// TIA Portal project "Erronka4" (V15.1)

(* hardware
DEVICE "S7-1200 station_1"  S7-1200 Station
   slot 0: "Rack_0"  S7-1200 Rack  Rack  V1.0
   slot 1: "PLC_1"  CPU 1214C AC/DC/Rly  6ES7 214-1BG40-0XB0  V4.0
   slot 3: "AQ 1x12BIT_1"  AQ1 signal board  6ES7 232-4HA30-0XB0  V1.0
*)

// ===== PLC "PLC_1"  CPU 1214C AC/DC/Rly =====

VAR_GLOBAL   // PLC tag table "Etapas"
   "Etapa0" AT %M16.0 : Bool;
   "Etapa1" AT %M16.1 : Bool;
   "Etapa2" AT %M16.2 : Bool;
   "Etapa3" AT %M16.3 : Bool;
   "Etapa4" AT %M16.4 : Bool;
   "Etapa5" AT %M16.5 : Bool;
   "Etapa6" AT %M16.6 : Bool;
   "Etapa7" AT %M16.7 : Bool;
   "Etapa8" AT %M17.0 : Bool;
   "Etapa9" AT %M17.1 : Bool;
   "Etapa20" AT %M20.0 : Bool;   // Inicio de STOP
   "Etapa21" AT %M20.1 : Bool;   // STOP
   "Etapa22" AT %M20.2 : Bool;   // STOP
   "MRMarca" AT %M90.0 : Bool;
   "Tag_2" AT %M302.0 : Bool;
   "Tag_3" AT %M300.0 : Bool;
   "Tag_4" AT %M300.1 : Bool;
   "Tag_6" AT %M301.0 : Bool;
   "Tag_7" AT %MB302 : Byte;
   "Tag_8" AT %MD16 : DWord;
   "Tag_9" AT %MD90 : DWord;
   "Tag_10" AT %M50.0 : Bool;
   "Tag_12" AT %M50.1 : Bool;
   "Tag_13" AT %MD70 : DWord;   // Tensión para mover MR
   "Tag_14" AT %MD74 : DWord;
   "CONTADORSALIDA" AT %MW100 : Int;
   "MARCAMOTORT" AT %M250.0 : Bool;
   "Tag_1" AT %MD250 : DWord;
END_VAR

VAR_GLOBAL   // PLC tag table "Entradas"
   "SDP1" AT %I0.1 : Bool;
   "SDP2" AT %I0.2 : Bool;
   "SDP3" AT %I0.3 : Bool;
   "SDP4" AT %I0.4 : Bool;
   "M" AT %I0.5 : Bool;
   "PE" AT %I0.6 : Bool;
   "CR0" AT %I0.7 : Bool;
   "CR1" AT %I1.0 : Bool;
   "CT0" AT %I1.1 : Bool;
   "CT1" AT %I1.2 : Bool;
   "CC0" AT %I1.3 : Bool;
   "CC1" AT %I1.4 : Bool;
   "STOP" AT %I0.0 : Bool;
END_VAR

VAR_GLOBAL   // PLC tag table "Salidas"
   "MR" AT %Q2.4 : Bool;
   "ACC" AT %Q0.1 : Bool;
   "DEC" AT %Q0.2 : Bool;
   "CR+" AT %Q0.3 : Bool;
   "CR-" AT %Q0.4 : Bool;
   "CT+" AT %Q0.5 : Bool;
   "CT-" AT %Q0.6 : Bool;
   "CC+" AT %Q0.7 : Bool;
   "CC-" AT %Q1.0 : Bool;
   "MT" AT %Q1.1 : Bool;
   "SEÑAL VARIADOR" AT %Q0.0 : Bool;
   "Tag_16" AT %QW80 : Int;
END_VAR

// folder: System blocks/Program resources

DATA_BLOCK "Temporizador1"   // DB1
{ S7_Optimized_Access := 'TRUE' }
AUTHOR : Simatic
FAMILY : IEC
NAME : IEC_TMR
VERSION : 1.0
// stored: InstanceOfName IEC_TIMER
"IEC_TIMER"
BEGIN
END_DATA_BLOCK

DATA_BLOCK "Contador"   // DB3
{ S7_Optimized_Access := 'TRUE' }
AUTHOR : Simatic
FAMILY : IEC
NAME : CNTR
VERSION : 1.0
// stored: InstanceOfName IEC_COUNTER
"IEC_COUNTER"
BEGIN
END_DATA_BLOCK

// folder: (top level)

FUNCTION "GrafcetPrincipal" : Void   // FC1, LAD
{ S7_Optimized_Access := 'TRUE' }
VERSION : 0.1
   VAR_TEMP   // added for the SCL form of the ladder/FBD networks
      _w1 : Bool;
   END_VAR
BEGIN

REGION Network 1
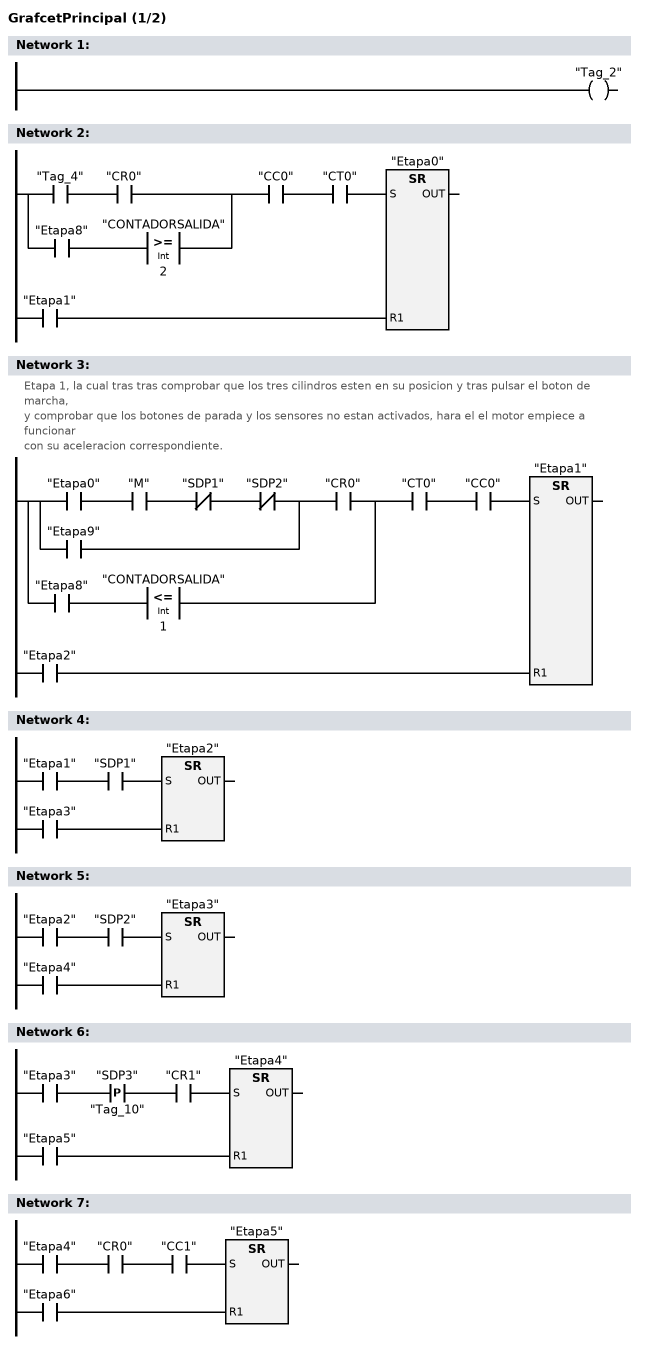
   RUNG wire#powerrail
      Coil( "Tag_2" )
   END_RUNG
   // the same network as SCL:
   "Tag_2" := TRUE;
END_REGION

REGION Network 2
   RUNG wire#powerrail
      Contact( "Tag_4" )
      Contact( "CR0" )
      wire#w1
      Contact( "CC0" )
      Contact( "CT0" )
      S_SR(operand := "Etapa0", r1 := wire#w2)
   END_RUNG
   RUNG wire#powerrail
      Contact( "Etapa8" )
      { S7_Templates := "SrcType := Int" } GE_Contact(in1 := "CONTADORSALIDA", in2 := 2)
   END_RUNG wire#w1
   RUNG wire#powerrail
      Contact( "Etapa1" )
   END_RUNG wire#w2
   // the same network as SCL:
   IF (("Tag_4" AND "CR0") OR ("Etapa8" AND ("CONTADORSALIDA" >= 2))) AND "CC0" AND "CT0" THEN
       "Etapa0" := TRUE;   // SR flip-flop
   END_IF;
   IF "Etapa1" THEN "Etapa0" := FALSE; END_IF;
END_REGION

REGION Network 3
   // Etapa 1, la cual tras tras comprobar que los tres cilindros esten en su posicion y tras pulsar el boton de marcha, 
   // y comprobar que los botones de parada y los sensores no estan activados, hara el el motor empiece a funcionar
   // con su aceleracion correspondiente.
   RUNG wire#powerrail
      Contact( "Etapa0" )
      Contact( "M" )
      I_Contact( "SDP1" )
      I_Contact( "SDP2" )
      wire#w1
      Contact( "CR0" )
      wire#w2
      Contact( "CT0" )
      Contact( "CC0" )
      S_SR(operand := "Etapa1", r1 := wire#w3)
   END_RUNG
   RUNG wire#powerrail
      Contact( "Etapa9" )
   END_RUNG wire#w1
   RUNG wire#powerrail
      Contact( "Etapa8" )
      { S7_Templates := "SrcType := Int" } LE_Contact(in1 := "CONTADORSALIDA", in2 := 1)
   END_RUNG wire#w2
   RUNG wire#powerrail
      Contact( "Etapa2" )
   END_RUNG wire#w3
   // the same network as SCL:
   IF (((("Etapa0" AND "M" AND NOT "SDP1" AND NOT "SDP2") OR "Etapa9") AND "CR0") OR ("Etapa8" AND ("CONTADORSALIDA" <= 1))) AND "CT0" AND "CC0" THEN
       "Etapa1" := TRUE;   // SR flip-flop
   END_IF;
   IF "Etapa2" THEN "Etapa1" := FALSE; END_IF;
END_REGION

REGION Network 4
   RUNG wire#powerrail
      Contact( "Etapa1" )
      Contact( "SDP1" )
      S_SR(operand := "Etapa2", r1 := wire#w1)
   END_RUNG
   RUNG wire#powerrail
      Contact( "Etapa3" )
   END_RUNG wire#w1
   // the same network as SCL:
   IF "Etapa1" AND "SDP1" THEN
       "Etapa2" := TRUE;   // SR flip-flop
   END_IF;
   IF "Etapa3" THEN "Etapa2" := FALSE; END_IF;
END_REGION

REGION Network 5
   RUNG wire#powerrail
      Contact( "Etapa2" )
      Contact( "SDP2" )
      S_SR(operand := "Etapa3", r1 := wire#w1)
   END_RUNG
   RUNG wire#powerrail
      Contact( "Etapa4" )
   END_RUNG wire#w1
   // the same network as SCL:
   IF "Etapa2" AND "SDP2" THEN
       "Etapa3" := TRUE;   // SR flip-flop
   END_IF;
   IF "Etapa4" THEN "Etapa3" := FALSE; END_IF;
END_REGION

REGION Network 6
   RUNG wire#powerrail
      Contact( "Etapa3" )
      P_Contact(operand := "SDP3", bit := "Tag_10")
      Contact( "CR1" )
      S_SR(operand := "Etapa4", r1 := wire#w1)
   END_RUNG
   RUNG wire#powerrail
      Contact( "Etapa5" )
   END_RUNG wire#w1
   // the same network as SCL:
   #_w1 := "Etapa3" AND "SDP3" AND NOT "Tag_10";   // rising edge of "SDP3"
   "Tag_10" := "SDP3";
   IF #_w1 AND "CR1" THEN
       "Etapa4" := TRUE;   // SR flip-flop
   END_IF;
   IF "Etapa5" THEN "Etapa4" := FALSE; END_IF;
END_REGION

REGION Network 7
   RUNG wire#powerrail
      Contact( "Etapa4" )
      Contact( "CR0" )
      Contact( "CC1" )
      S_SR(operand := "Etapa5", r1 := wire#w1)
   END_RUNG
   RUNG wire#powerrail
      Contact( "Etapa6" )
   END_RUNG wire#w1
   // the same network as SCL:
   IF "Etapa4" AND "CR0" AND "CC1" THEN
       "Etapa5" := TRUE;   // SR flip-flop
   END_IF;
   IF "Etapa6" THEN "Etapa5" := FALSE; END_IF;
END_REGION

REGION Network 8
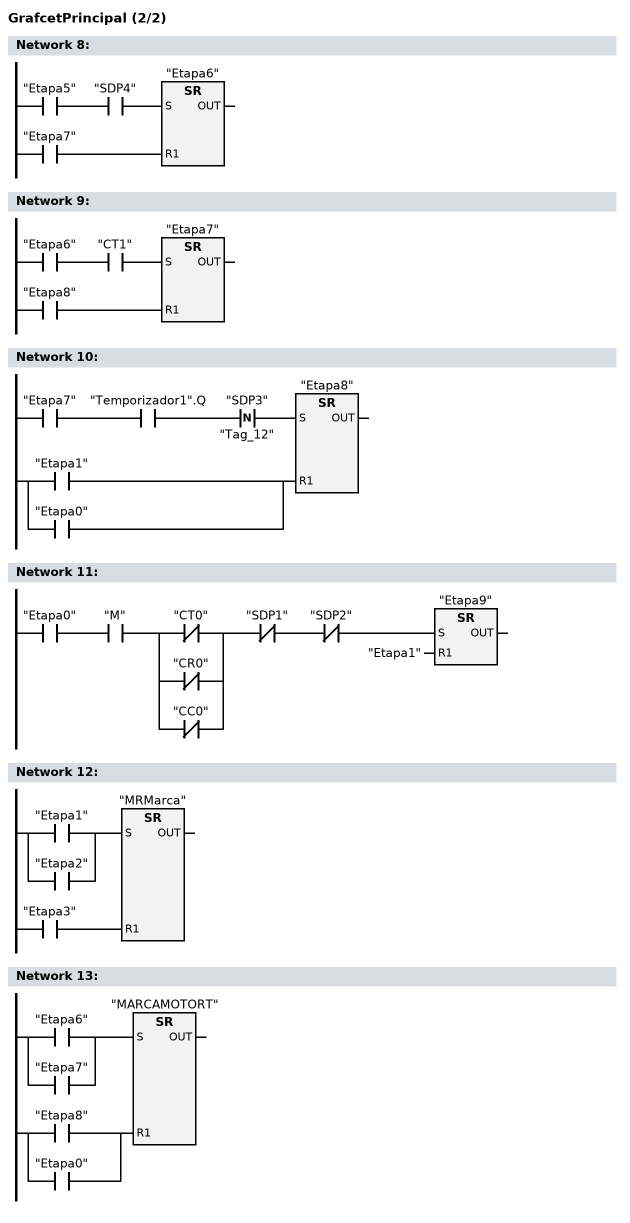
   RUNG wire#powerrail
      Contact( "Etapa5" )
      Contact( "SDP4" )
      S_SR(operand := "Etapa6", r1 := wire#w1)
   END_RUNG
   RUNG wire#powerrail
      Contact( "Etapa7" )
   END_RUNG wire#w1
   // the same network as SCL:
   IF "Etapa5" AND "SDP4" THEN
       "Etapa6" := TRUE;   // SR flip-flop
   END_IF;
   IF "Etapa7" THEN "Etapa6" := FALSE; END_IF;
END_REGION

REGION Network 9
   RUNG wire#powerrail
      Contact( "Etapa6" )
      Contact( "CT1" )
      S_SR(operand := "Etapa7", r1 := wire#w1)
   END_RUNG
   RUNG wire#powerrail
      Contact( "Etapa8" )
   END_RUNG wire#w1
   // the same network as SCL:
   IF "Etapa6" AND "CT1" THEN
       "Etapa7" := TRUE;   // SR flip-flop
   END_IF;
   IF "Etapa8" THEN "Etapa7" := FALSE; END_IF;
END_REGION

REGION Network 10
   RUNG wire#powerrail
      Contact( "Etapa7" )
      Contact( "Temporizador1".Q )
      N_Contact(operand := "SDP3", bit := "Tag_12")
      S_SR(operand := "Etapa8", r1 := wire#w1)
   END_RUNG
   RUNG wire#powerrail
      Contact( "Etapa1" )
   END_RUNG wire#w1
   RUNG wire#powerrail
      Contact( "Etapa0" )
   END_RUNG wire#w1
   // the same network as SCL:
   #_w1 := "Etapa7" AND "Temporizador1".Q AND NOT "SDP3" AND "Tag_12";   // falling edge of "SDP3"
   "Tag_12" := "SDP3";
   IF #_w1 THEN
       "Etapa8" := TRUE;   // SR flip-flop
   END_IF;
   IF "Etapa1" OR "Etapa0" THEN "Etapa8" := FALSE; END_IF;
END_REGION

REGION Network 11
   RUNG wire#powerrail
      Contact( "Etapa0" )
      Contact( "M" )
      wire#w1
      I_Contact( "CT0" )
      wire#w2
      I_Contact( "SDP1" )
      I_Contact( "SDP2" )
      S_SR(operand := "Etapa9", r1 := "Etapa1")
   END_RUNG
   RUNG wire#w1
      I_Contact( "CR0" )
   END_RUNG wire#w2
   RUNG wire#w1
      I_Contact( "CC0" )
   END_RUNG wire#w2
   // the same network as SCL:
   IF "Etapa0" AND "M" AND (NOT "CT0" OR NOT "CR0" OR NOT "CC0") AND NOT "SDP1" AND NOT "SDP2" THEN
       "Etapa9" := TRUE;   // SR flip-flop
   END_IF;
   IF "Etapa1" THEN "Etapa9" := FALSE; END_IF;
END_REGION

REGION Network 12
   RUNG wire#powerrail
      Contact( "Etapa1" )
      wire#w1
      S_SR(operand := "MRMarca", r1 := wire#w2)
   END_RUNG
   RUNG wire#powerrail
      Contact( "Etapa2" )
   END_RUNG wire#w1
   RUNG wire#powerrail
      Contact( "Etapa3" )
   END_RUNG wire#w2
   // the same network as SCL:
   IF "Etapa1" OR "Etapa2" THEN
       "MRMarca" := TRUE;   // SR flip-flop
   END_IF;
   IF "Etapa3" THEN "MRMarca" := FALSE; END_IF;
END_REGION

REGION Network 13
   RUNG wire#powerrail
      Contact( "Etapa6" )
      wire#w1
      S_SR(operand := "MARCAMOTORT", r1 := wire#w2)
   END_RUNG
   RUNG wire#powerrail
      Contact( "Etapa7" )
   END_RUNG wire#w1
   RUNG wire#powerrail
      Contact( "Etapa8" )
   END_RUNG wire#w2
   RUNG wire#powerrail
      Contact( "Etapa0" )
   END_RUNG wire#w2
   // the same network as SCL:
   IF "Etapa6" OR "Etapa7" THEN
       "MARCAMOTORT" := TRUE;   // SR flip-flop
   END_IF;
   IF "Etapa8" OR "Etapa0" THEN "MARCAMOTORT" := FALSE; END_IF;
END_REGION
END_FUNCTION

FUNCTION "ParadaStop" : Void   // FC2, LAD
{ S7_Optimized_Access := 'TRUE' }
VERSION : 0.1
BEGIN

REGION Network 1
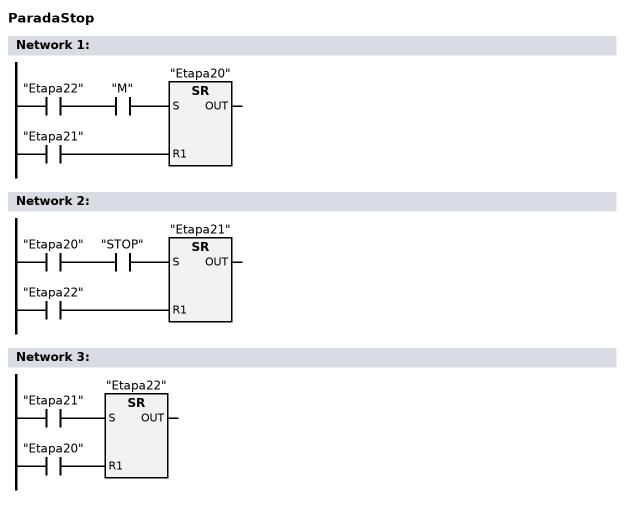
   RUNG wire#powerrail
      Contact( "Etapa22" )
      Contact( "M" )
      S_SR(operand := "Etapa20", r1 := wire#w1)
   END_RUNG
   RUNG wire#powerrail
      Contact( "Etapa21" )
   END_RUNG wire#w1
   // the same network as SCL:
   IF "Etapa22" AND "M" THEN
       "Etapa20" := TRUE;   // SR flip-flop
   END_IF;
   IF "Etapa21" THEN "Etapa20" := FALSE; END_IF;
END_REGION

REGION Network 2
   RUNG wire#powerrail
      Contact( "Etapa20" )
      Contact( "STOP" )
      S_SR(operand := "Etapa21", r1 := wire#w1)
   END_RUNG
   RUNG wire#powerrail
      Contact( "Etapa22" )
   END_RUNG wire#w1
   // the same network as SCL:
   IF "Etapa20" AND "STOP" THEN
       "Etapa21" := TRUE;   // SR flip-flop
   END_IF;
   IF "Etapa22" THEN "Etapa21" := FALSE; END_IF;
END_REGION

REGION Network 3
   RUNG wire#powerrail
      Contact( "Etapa21" )
      S_SR(operand := "Etapa22", r1 := wire#w1)
   END_RUNG
   RUNG wire#powerrail
      Contact( "Etapa20" )
   END_RUNG wire#w1
   // the same network as SCL:
   IF "Etapa21" THEN
       "Etapa22" := TRUE;   // SR flip-flop
   END_IF;
   IF "Etapa20" THEN "Etapa22" := FALSE; END_IF;
END_REGION
END_FUNCTION

FUNCTION "ParadaEmergencia" : Void   // FC3, LAD
{ S7_Optimized_Access := 'TRUE' }
VERSION : 0.1
BEGIN

REGION Network 1
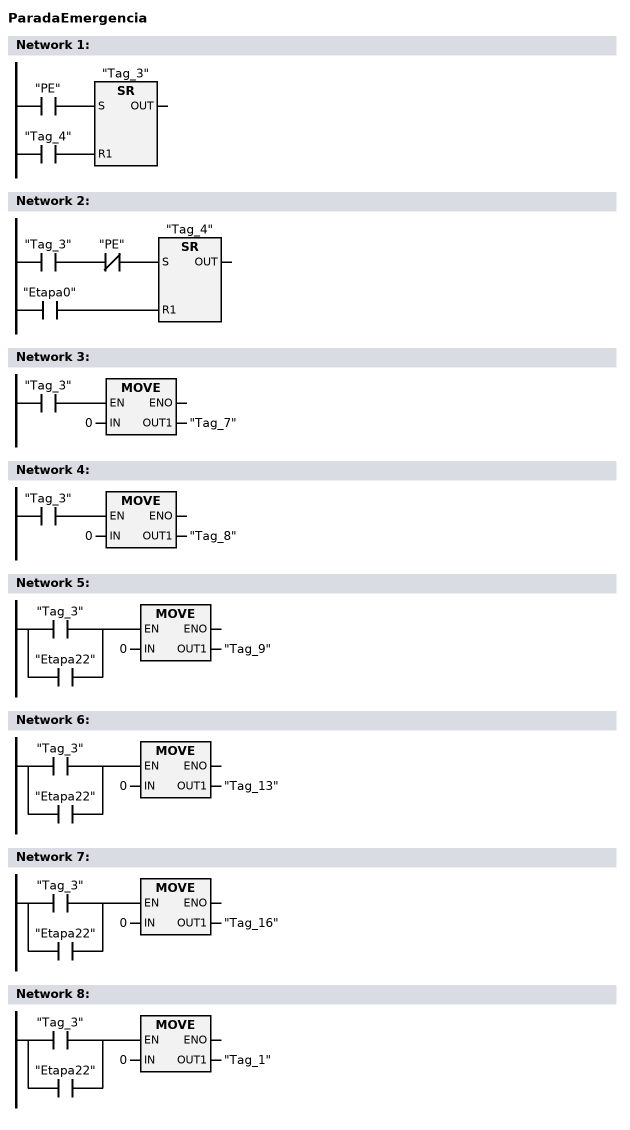
   RUNG wire#powerrail
      Contact( "PE" )
      S_SR(operand := "Tag_3", r1 := wire#w1)
   END_RUNG
   RUNG wire#powerrail
      Contact( "Tag_4" )
   END_RUNG wire#w1
   // the same network as SCL:
   IF "PE" THEN
       "Tag_3" := TRUE;   // SR flip-flop
   END_IF;
   IF "Tag_4" THEN "Tag_3" := FALSE; END_IF;
END_REGION

REGION Network 2
   RUNG wire#powerrail
      Contact( "Tag_3" )
      I_Contact( "PE" )
      S_SR(operand := "Tag_4", r1 := wire#w1)
   END_RUNG
   RUNG wire#powerrail
      Contact( "Etapa0" )
   END_RUNG wire#w1
   // the same network as SCL:
   IF "Tag_3" AND NOT "PE" THEN
       "Tag_4" := TRUE;   // SR flip-flop
   END_IF;
   IF "Etapa0" THEN "Tag_4" := FALSE; END_IF;
END_REGION

REGION Network 3
   RUNG wire#powerrail
      Contact( "Tag_3" )
      Move(in := 0, out1 => "Tag_7")
   END_RUNG
   // the same network as SCL:
   IF "Tag_3" THEN "Tag_7" := 0; END_IF;
END_REGION

REGION Network 4
   RUNG wire#powerrail
      Contact( "Tag_3" )
      Move(in := 0, out1 => "Tag_8")
   END_RUNG
   // the same network as SCL:
   IF "Tag_3" THEN "Tag_8" := 0; END_IF;
END_REGION

REGION Network 5
   RUNG wire#powerrail
      Contact( "Tag_3" )
      wire#w1
      Move(in := 0, out1 => "Tag_9")
   END_RUNG
   RUNG wire#powerrail
      Contact( "Etapa22" )
   END_RUNG wire#w1
   // the same network as SCL:
   IF "Tag_3" OR "Etapa22" THEN "Tag_9" := 0; END_IF;
END_REGION

REGION Network 6
   RUNG wire#powerrail
      Contact( "Tag_3" )
      wire#w1
      Move(in := 0, out1 => "Tag_13")
   END_RUNG
   RUNG wire#powerrail
      Contact( "Etapa22" )
   END_RUNG wire#w1
   // the same network as SCL:
   IF "Tag_3" OR "Etapa22" THEN "Tag_13" := 0; END_IF;
END_REGION

REGION Network 7
   RUNG wire#powerrail
      Contact( "Tag_3" )
      wire#w1
      Move(in := 0, out1 => "Tag_16")
   END_RUNG
   RUNG wire#powerrail
      Contact( "Etapa22" )
   END_RUNG wire#w1
   // the same network as SCL:
   IF "Tag_3" OR "Etapa22" THEN "Tag_16" := 0; END_IF;
END_REGION

REGION Network 8
   RUNG wire#powerrail
      Contact( "Tag_3" )
      wire#w1
      Move(in := 0, out1 => "Tag_1")
   END_RUNG
   RUNG wire#powerrail
      Contact( "Etapa22" )
   END_RUNG wire#w1
   // the same network as SCL:
   IF "Tag_3" OR "Etapa22" THEN "Tag_1" := 0; END_IF;
END_REGION
END_FUNCTION

FUNCTION "Salidas" : Void   // FC4, LAD
{ S7_Optimized_Access := 'TRUE' }
VERSION : 0.1
BEGIN

REGION Network 1
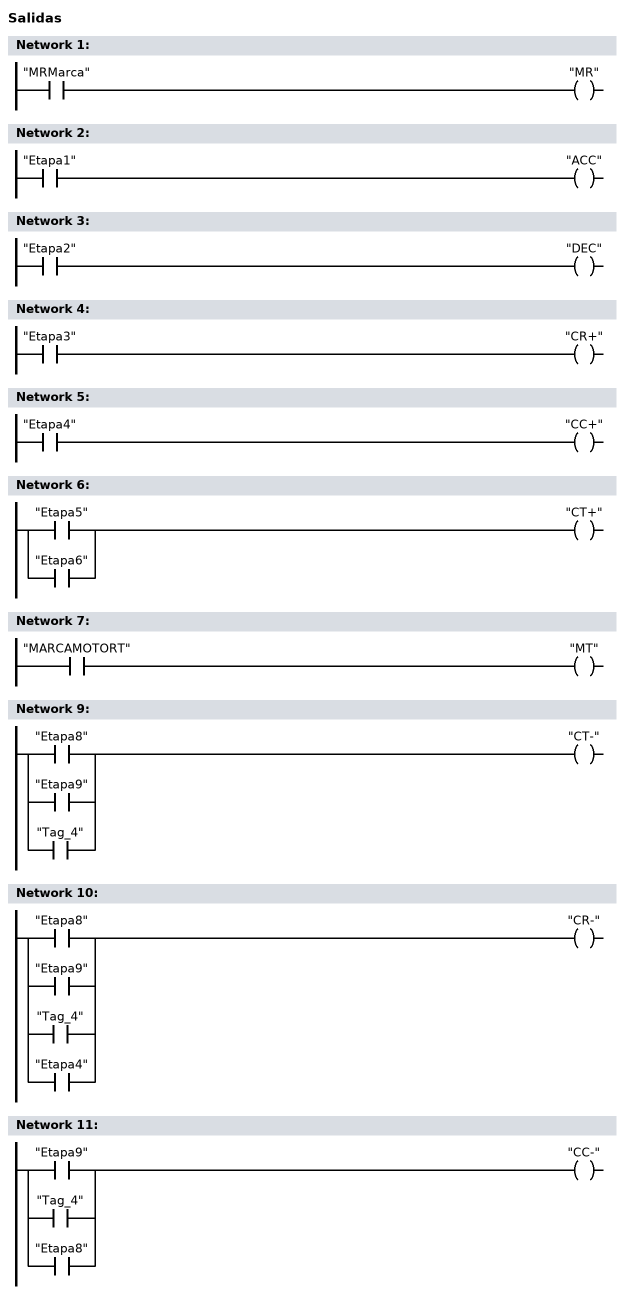
   RUNG wire#powerrail
      Contact( "MRMarca" )
      Coil( "MR" )
   END_RUNG
   // the same network as SCL:
   "MR" := "MRMarca";
END_REGION

REGION Network 2
   RUNG wire#powerrail
      Contact( "Etapa1" )
      Coil( "ACC" )
   END_RUNG
   // the same network as SCL:
   "ACC" := "Etapa1";
END_REGION

REGION Network 3
   RUNG wire#powerrail
      Contact( "Etapa2" )
      Coil( "DEC" )
   END_RUNG
   // the same network as SCL:
   "DEC" := "Etapa2";
END_REGION

REGION Network 4
   RUNG wire#powerrail
      Contact( "Etapa3" )
      Coil( "CR+" )
   END_RUNG
   // the same network as SCL:
   "CR+" := "Etapa3";
END_REGION

REGION Network 5
   RUNG wire#powerrail
      Contact( "Etapa4" )
      Coil( "CC+" )
   END_RUNG
   // the same network as SCL:
   "CC+" := "Etapa4";
END_REGION

REGION Network 6
   RUNG wire#powerrail
      Contact( "Etapa5" )
      wire#w1
      Coil( "CT+" )
   END_RUNG
   RUNG wire#powerrail
      Contact( "Etapa6" )
   END_RUNG wire#w1
   // the same network as SCL:
   "CT+" := "Etapa5" OR "Etapa6";
END_REGION

REGION Network 7
   RUNG wire#powerrail
      Contact( "MARCAMOTORT" )
      Coil( "MT" )
   END_RUNG
   // the same network as SCL:
   "MT" := "MARCAMOTORT";
END_REGION

REGION Network 9
   RUNG wire#powerrail
      Contact( "Etapa8" )
      wire#w1
      Coil( "CT-" )
   END_RUNG
   RUNG wire#powerrail
      Contact( "Etapa9" )
   END_RUNG wire#w1
   RUNG wire#powerrail
      Contact( "Tag_4" )
   END_RUNG wire#w1
   // the same network as SCL:
   "CT-" := "Etapa8" OR "Etapa9" OR "Tag_4";
END_REGION

REGION Network 10
   RUNG wire#powerrail
      Contact( "Etapa8" )
      wire#w1
      Coil( "CR-" )
   END_RUNG
   RUNG wire#powerrail
      Contact( "Etapa9" )
   END_RUNG wire#w1
   RUNG wire#powerrail
      Contact( "Tag_4" )
   END_RUNG wire#w1
   RUNG wire#powerrail
      Contact( "Etapa4" )
   END_RUNG wire#w1
   // the same network as SCL:
   "CR-" := "Etapa8" OR "Etapa9" OR "Tag_4" OR "Etapa4";
END_REGION

REGION Network 11
   RUNG wire#powerrail
      Contact( "Etapa9" )
      wire#w1
      Coil( "CC-" )
   END_RUNG
   RUNG wire#powerrail
      Contact( "Tag_4" )
   END_RUNG wire#w1
   RUNG wire#powerrail
      Contact( "Etapa8" )
   END_RUNG wire#w1
   // the same network as SCL:
   "CC-" := "Etapa9" OR "Tag_4" OR "Etapa8";
END_REGION
END_FUNCTION

FUNCTION "Temporizador" : Void   // FC5, LAD
{ S7_Optimized_Access := 'TRUE' }
VERSION : 0.1
BEGIN

REGION Network 1
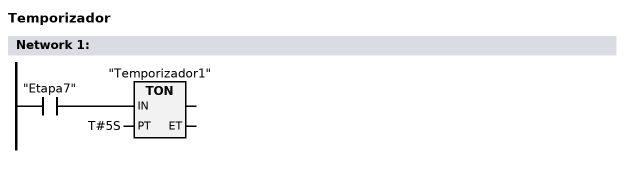
   "Temporizador1".TON(IN := "Etapa7", PT := T#5S);
END_REGION
END_FUNCTION

FUNCTION "Contadores" : Void   // FC6, LAD
{ S7_Optimized_Access := 'TRUE' }
VERSION : 0.1
BEGIN

REGION Network 1
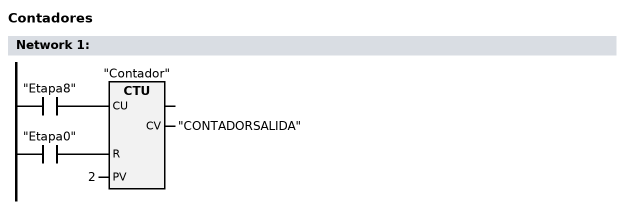
   "Contador".CTU(CU := "Etapa8", R := "Etapa0", PV := 2, CV => "CONTADORSALIDA");
END_REGION
END_FUNCTION

FUNCTION "Variador de Velocidad" : Void   // FC7, LAD
{ S7_Optimized_Access := 'TRUE' }
VERSION : 0.1
BEGIN

REGION Network 1
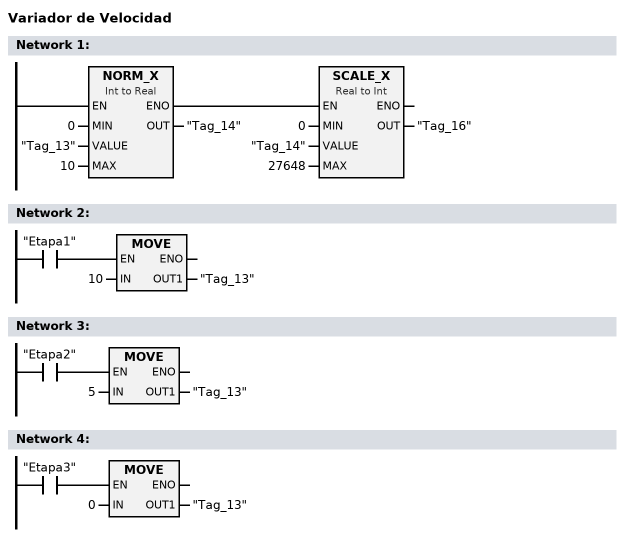
   RUNG wire#powerrail
      { S7_Templates := "[SrcType := Int, DestType := Real]" } Normalize(min := 0, value := "Tag_13", max := 10, out => "Tag_14")
      { S7_Templates := "[SrcType := Real, DestType := Int]" } Scale(min := 0, value := "Tag_14", max := 27648, out => "Tag_16")
   END_RUNG
   // the same network as SCL:
   "Tag_14" := NORM_X(MIN := 0, VALUE := "Tag_13", MAX := 10);
   "Tag_16" := SCALE_X(MIN := 0, VALUE := "Tag_14", MAX := 27648);
END_REGION

REGION Network 2
   RUNG wire#powerrail
      Contact( "Etapa1" )
      Move(in := 10, out1 => "Tag_13")
   END_RUNG
   // the same network as SCL:
   IF "Etapa1" THEN "Tag_13" := 10; END_IF;
END_REGION

REGION Network 3
   RUNG wire#powerrail
      Contact( "Etapa2" )
      Move(in := 5, out1 => "Tag_13")
   END_RUNG
   // the same network as SCL:
   IF "Etapa2" THEN "Tag_13" := 5; END_IF;
END_REGION

REGION Network 4
   RUNG wire#powerrail
      Contact( "Etapa3" )
      Move(in := 0, out1 => "Tag_13")
   END_RUNG
   // the same network as SCL:
   IF "Etapa3" THEN "Tag_13" := 0; END_IF;
END_REGION
END_FUNCTION

FUNCTION "AcDecVariador" : Void   // FC8, LAD
{ S7_Optimized_Access := 'TRUE' }
VERSION : 0.1
BEGIN

REGION Network 1
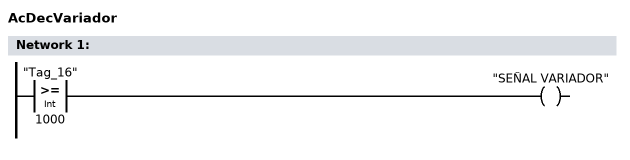
   RUNG wire#powerrail
      { S7_Templates := "SrcType := Int" } GE_Contact(in1 := "Tag_16", in2 := 1000)
      Coil( "SEÑAL VARIADOR" )
   END_RUNG
   // the same network as SCL:
   "SEÑAL VARIADOR" := "Tag_16" >= 1000;
END_REGION
END_FUNCTION

ORGANIZATION_BLOCK "Main"   // OB1, LAD, ProgramCycle
TITLE = "Main Program Sweep (Cycle)"
{ S7_Optimized_Access := 'TRUE' }
VERSION : 0.1
   VAR_INPUT
      Initial_Call : Bool;   // Initial call of this OB
      Remanence : Bool;   // =True, if remanent data are available
   END_VAR
BEGIN

REGION Network 1
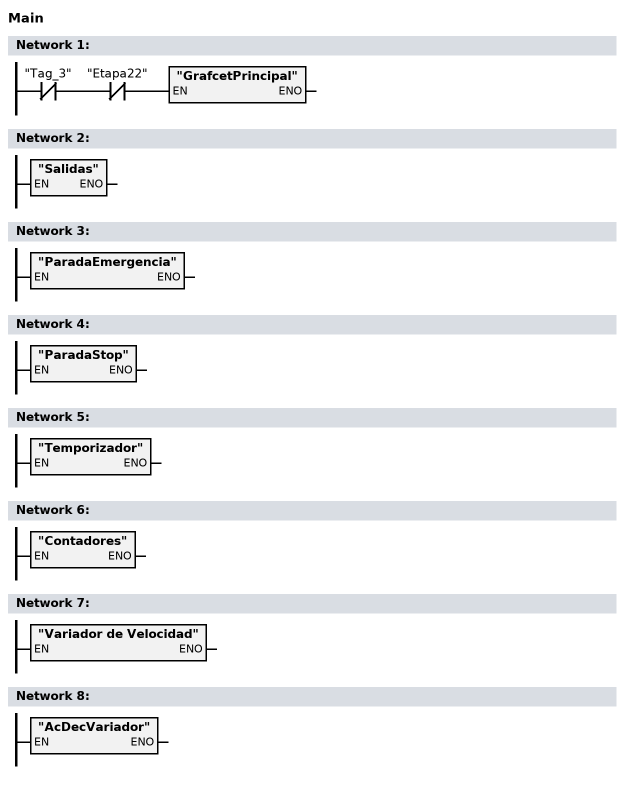
   RUNG wire#powerrail
      I_Contact( "Tag_3" )
      I_Contact( "Etapa22" )
      "GrafcetPrincipal"()
   END_RUNG
   // the same network as SCL:
   IF NOT "Tag_3" AND NOT "Etapa22" THEN "GrafcetPrincipal"(); END_IF;
END_REGION

REGION Network 2
   RUNG wire#powerrail
      "Salidas"()
   END_RUNG
   // the same network as SCL:
   "Salidas"();
END_REGION

REGION Network 3
   RUNG wire#powerrail
      "ParadaEmergencia"()
   END_RUNG
   // the same network as SCL:
   "ParadaEmergencia"();
END_REGION

REGION Network 4
   RUNG wire#powerrail
      "ParadaStop"()
   END_RUNG
   // the same network as SCL:
   "ParadaStop"();
END_REGION

REGION Network 5
   RUNG wire#powerrail
      "Temporizador"()
   END_RUNG
   // the same network as SCL:
   "Temporizador"();
END_REGION

REGION Network 6
   RUNG wire#powerrail
      "Contadores"()
   END_RUNG
   // the same network as SCL:
   "Contadores"();
END_REGION

REGION Network 7
   RUNG wire#powerrail
      "Variador de Velocidad"()
   END_RUNG
   // the same network as SCL:
   "Variador de Velocidad"();
END_REGION

REGION Network 8
   RUNG wire#powerrail
      "AcDecVariador"()
   END_RUNG
   // the same network as SCL:
   "AcDecVariador"();
END_REGION
END_ORGANIZATION_BLOCK

ORGANIZATION_BLOCK "Startup"   // OB100, LAD, Startup
TITLE = "Complete Restart"
{ S7_Optimized_Access := 'TRUE' }
VERSION : 0.1
   VAR_INPUT
      LostRetentive : Bool;   // True if retentive data are lost
      LostRTC : Bool;   // True if date and time are lost
   END_VAR
BEGIN

REGION Network 1
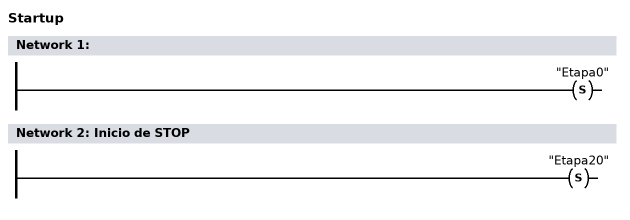
   RUNG wire#powerrail
      S_Coil( "Etapa0" )
   END_RUNG
   // the same network as SCL:
   "Etapa0" := TRUE;
END_REGION

REGION Network 2: Inicio de STOP
   RUNG wire#powerrail
      S_Coil( "Etapa20" )
   END_RUNG
   // the same network as SCL:
   "Etapa20" := TRUE;
END_REGION
END_ORGANIZATION_BLOCK